# EPICS alarm handler configuration: mps_database/bareTest/alarms/areas/mpln_bpn23_mp01.alhConfig
GROUP NULL MPLN:BPN23:MP01:1
$ALIAS MPS Link Node 87
$GUIDANCE
LTUH MPS
   Group Name: MPLN:BPN23:MP01:1
   Summary PV:  MPLN:BPN23:MP01:1:STATSUMY
$END
CHANNEL  MPLN:BPN23:MP01:1    MPLN:BPN23:MP01:1:MPS_EN_RBV		-----
CHANNEL  MPLN:BPN23:MP01:1    MPLN:BPN23:MP01:1:LC1_MODE_RBV		-----
